SYSTEM TEST_SWING (* Test of Swing components *)
  (* Standard: 61499-1 *)
  (* Version 0.0, 2004-06-18, JHC, Rockwell Automation *)
  APPLICATION APP1
  END_APPLICATION
  DEVICE DEV1 : FRAME_DEVICE(BOUNDS := [100,100,250,225], GRID := [7,1])
    RESOURCE RES1 : PANEL_RESOURCE
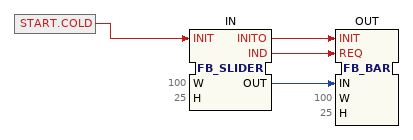
      FBS
        IN : FB_SLIDER(W := 100, H := 25);
        OUT : FB_BAR(W := 100, H := 25);
      END_FBS
      EVENT_CONNECTIONS
        START.COLD TO IN.INIT;
        IN.INITO TO OUT.INIT;
        IN.IND TO OUT.REQ;
      END_CONNECTIONS
      DATA_CONNECTIONS
        IN.OUT TO OUT.IN;
      END_CONNECTIONS
    END_RESOURCE
    RESOURCE RES2 : PANEL_RESOURCE
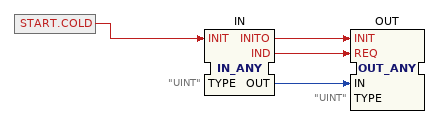
      FBS
        IN : IN_ANY(TYPE := "UINT");
        OUT : OUT_ANY(TYPE := "UINT");
      END_FBS
      EVENT_CONNECTIONS
        START.COLD TO IN.INIT;
        IN.INITO TO OUT.INIT;
        IN.IND TO OUT.REQ;
      END_CONNECTIONS
      DATA_CONNECTIONS
        IN.OUT TO OUT.IN;
      END_CONNECTIONS
    END_RESOURCE
    RESOURCE RES3 : PANEL_RESOURCE
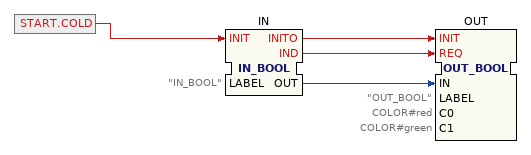
      FBS
        IN : IN_BOOL(LABEL := "IN_BOOL");
        OUT : OUT_BOOL(LABEL := "OUT_BOOL", C0 := COLOR#red, C1 := COLOR#green);
      END_FBS
      EVENT_CONNECTIONS
        START.COLD TO IN.INIT;
        IN.INITO TO OUT.INIT;
        IN.IND TO OUT.REQ;
      END_CONNECTIONS
      DATA_CONNECTIONS
        IN.OUT TO OUT.IN;
      END_CONNECTIONS
    END_RESOURCE
    RESOURCE RES4 : PANEL_RESOURCE
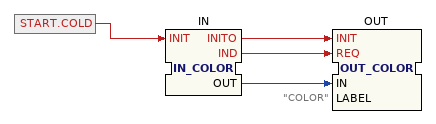
      FBS
        IN : IN_COLOR;
        OUT : OUT_COLOR(LABEL := "COLOR");
      END_FBS
      EVENT_CONNECTIONS
        START.COLD TO IN.INIT;
        IN.INITO TO OUT.INIT;
        IN.IND TO OUT.REQ;
      END_CONNECTIONS
      DATA_CONNECTIONS
        IN.OUT TO OUT.IN;
      END_CONNECTIONS
    END_RESOURCE
    RESOURCE RES5 : PANEL_RESOURCE
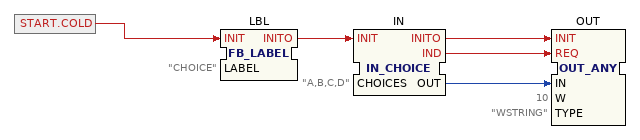
      FBS
        IN : IN_CHOICE(CHOICES := "A,B,C,D");
        OUT : OUT_ANY(W := 10, TYPE := "WSTRING");
        LBL : FB_LABEL(LABEL := "CHOICE");
      END_FBS
      EVENT_CONNECTIONS
        IN.INITO TO OUT.INIT;
        IN.IND TO OUT.REQ;
        START.COLD TO LBL.INIT;
        LBL.INITO TO IN.INIT;
      END_CONNECTIONS
      DATA_CONNECTIONS
        IN.OUT TO OUT.IN;
      END_CONNECTIONS
    END_RESOURCE
    RESOURCE RES6 : PANEL_RESOURCE
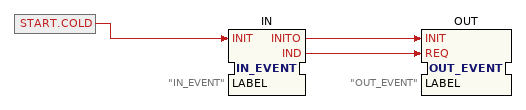
      FBS
        IN : IN_EVENT(LABEL := "IN_EVENT");
        OUT : OUT_EVENT(LABEL := "OUT_EVENT");
      END_FBS
      EVENT_CONNECTIONS
        START.COLD TO IN.INIT;
        IN.INITO TO OUT.INIT;
        IN.IND TO OUT.REQ;
      END_CONNECTIONS
    END_RESOURCE
    RESOURCE RES7 : PANEL_RESOURCE
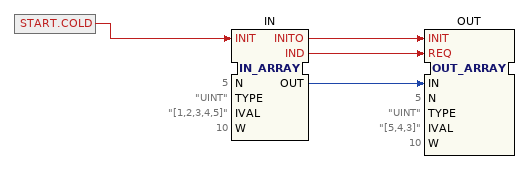
      FBS
        IN : IN_ARRAY(N := 5, TYPE := "UINT", IVAL := "[1,2,3,4,5]", W := 10);
        OUT : OUT_ARRAY(N := 5, TYPE := "UINT", IVAL := "[5,4,3]", W := 10);
      END_FBS
      EVENT_CONNECTIONS
        START.COLD TO IN.INIT;
        IN.INITO TO OUT.INIT;
        IN.IND TO OUT.REQ;
      END_CONNECTIONS
      DATA_CONNECTIONS
        IN.OUT TO OUT.IN;
      END_CONNECTIONS
    END_RESOURCE
  END_DEVICE
END_SYSTEM
